Universal Robots PolyScope program: mansion.urp

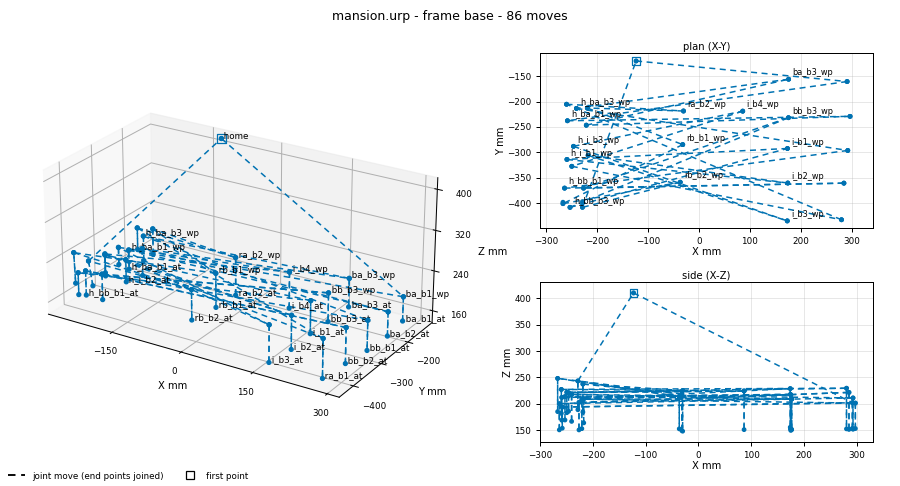
[picture p0: tool path of mansion.urp in frame base, 86 of 86 moves have a stored position in this frame; points joined in program order, loops and branches not executed]
Program mansion (installation=default directory=/programs/ITER createdIn=5.3.1.64192 lastSavedIn=5.3.1.64192 robotSerialNumber=20195300365)
Calibrated DH parameters: a=[-0.000093, -0.190649, -0.212673, 0.000091, -0.000205, 0]; d=[0.151591, 44.061648, -42.488068, -1.442789, 0.085322, 0.091911]; alpha=[1.570082, -0.003447, 0.007513, 1.572293, -1.571904, 0]; deltaTheta=[0, -0.672656, 0.728185, -0.055522, 0.000005, 0]
Robot Program (runOnlyOnce=true)
  URCap Gripper Activate (Robotiq_Grippers, Robotiq Inc.) dataModel(ResetAndActivateKey=false)
  URCap Gripper (Robotiq_Grippers, Robotiq Inc.) dataModel(position=50.0, force=100.0, speed=100.0, positionInDouble=50.0, forceInDouble=100.0, speedInDouble=100.0, slaveIds=[9], blocking=true)
  MoveJ speed 60 deg/s, acceleration 80 deg/s^2 (useActiveTCP=true) feature=Base
    Waypoint home: TCP in base x=-122.926 y=-120.377 z=410.038 mm, rx=2.273 ry=2.1657 rz=-0.0264 rad; joints [-85.876, -57.16, -80.452, -131.626, 89.649, -263.131] deg
  Folder Base_A
    MoveJ speed 60 deg/s, acceleration 80 deg/s^2 (useActiveTCP=true) feature=Base
      Waypoint ba_b1_wp: TCP in base x=291.339 y=-160.763 z=202.267 mm, rx=2.2196 ry=2.1634 rz=-0.046 rad; joints [-5.134, -97.09, -111.302, -60.85, 87.435, -183.275] deg
      Waypoint ba_b1_at: TCP in base x=291.327 y=-160.782 z=153.554 mm, rx=2.2196 ry=2.1633 rz=-0.046 rad; joints [-5.155, -104.362, -118.201, -46.683, 87.36, -183.222] deg
      URCap Gripper (Robotiq_Grippers, Robotiq Inc.) dataModel(position=100.0, force=100.0, speed=100.0, positionInDouble=100.0, forceInDouble=100.0, speedInDouble=100.0, slaveIds=[9], blocking=true)
      Waypoint ba_b1_wp: TCP in base x=291.339 y=-160.763 z=202.267 mm, rx=2.2196 ry=2.1634 rz=-0.046 rad; joints [-5.134, -97.09, -111.302, -60.85, 87.435, -183.275] deg
      Waypoint h_ba_b1_wp: TCP in base x=-257.858 y=-237.79 z=193.998 mm, rx=-3.1287 ry=0.0473 rz=-0.0059 rad; joints [-115.618, -102.966, -105.931, -61.783, 90.175, -203.494] deg
      Waypoint h_ba_b1_at: TCP in base x=-257.856 y=-237.787 z=153.878 mm, rx=-3.1287 ry=0.0473 rz=-0.006 rad; joints [-115.632, -108.549, -111.296, -50.837, 90.123, -203.451] deg
      URCap Gripper (Robotiq_Grippers, Robotiq Inc.) dataModel(position=50.0, force=100.0, speed=100.0, positionInDouble=50.0, forceInDouble=100.0, speedInDouble=100.0, slaveIds=[9], blocking=true)
      Waypoint h_ba_b1_wp: TCP in base x=-257.858 y=-237.79 z=193.998 mm, rx=-3.1287 ry=0.0473 rz=-0.0059 rad; joints [-115.618, -102.966, -105.931, -61.783, 90.175, -203.494] deg
    MoveJ speed 60 deg/s, acceleration 80 deg/s^2 (useActiveTCP=true) feature=Base
      Waypoint ba_b2_wp: TCP in base x=297.099 y=-229.137 z=201.509 mm, rx=2.2534 ry=2.1854 rz=-0.0426 rad; joints [-17.056, -107.569, -97.554, -65.462, 88.854, -194.942] deg
      Waypoint ba_b2_at: TCP in base x=297.093 y=-229.143 z=153.246 mm, rx=2.2534 ry=2.1854 rz=-0.0427 rad; joints [-17.073, -113.534, -103.963, -53.09, 88.799, -194.893] deg
      URCap Gripper (Robotiq_Grippers, Robotiq Inc.) dataModel(position=100.0, force=100.0, speed=100.0, positionInDouble=100.0, forceInDouble=100.0, speedInDouble=100.0, slaveIds=[9], blocking=true)
      Waypoint ba_b2_wp: TCP in base x=297.099 y=-229.137 z=201.509 mm, rx=2.2534 ry=2.1854 rz=-0.0426 rad; joints [-17.056, -107.569, -97.554, -65.462, 88.854, -194.942] deg
      Waypoint h_ba_b2_wp: TCP in base x=-220.82 y=-246.483 z=208.907 mm, rx=-3.1272 ry=0.0669 rz=0.002 rad; joints [-108.726, -96.552, -109.252, -64.858, 89.998, -195.885] deg
      Waypoint h_ba_b2_at: TCP in base x=-220.812 y=-246.497 z=153.058 mm, rx=-3.1273 ry=0.0669 rz=0.002 rad; joints [-108.744, -104.469, -117.433, -48.758, 89.918, -195.821] deg
      URCap Gripper (Robotiq_Grippers, Robotiq Inc.) dataModel(position=50.0, force=100.0, speed=100.0, positionInDouble=50.0, forceInDouble=100.0, speedInDouble=100.0, slaveIds=[9], blocking=true)
      Waypoint h_ba_b2_wp: TCP in base x=-220.82 y=-246.483 z=208.907 mm, rx=-3.1272 ry=0.0669 rz=0.002 rad; joints [-108.726, -96.552, -109.252, -64.858, 89.998, -195.885] deg
    MoveJ speed 60 deg/s, acceleration 80 deg/s^2 (useActiveTCP=true) feature=Base
      Waypoint ba_b3_wp: TCP in base x=176.479 y=-156.192 z=208.942 mm, rx=2.1987 ry=2.1726 rz=-0.0159 rad; joints [-7.147, -67.928, -134.317, -65.798, 88.131, -186.073] deg
      Waypoint ba_b3_at: TCP in base x=176.475 y=-156.198 z=150.955 mm, rx=2.1987 ry=2.1726 rz=-0.0159 rad; joints [-7.184, -79.69, -145.938, -42.419, 87.997, -185.98] deg
      URCap Gripper (Robotiq_Grippers, Robotiq Inc.) dataModel(position=100.0, force=100.0, speed=100.0, positionInDouble=100.0, forceInDouble=100.0, speedInDouble=100.0, slaveIds=[9], blocking=true)
      Waypoint ba_b3_wp: TCP in base x=176.479 y=-156.192 z=208.942 mm, rx=2.1987 ry=2.1726 rz=-0.0159 rad; joints [-7.147, -67.928, -134.317, -65.798, 88.131, -186.073] deg
      Waypoint h_ba_b3_wp: TCP in base x=-240.197 y=-213.51 z=217.855 mm, rx=2.242 ry=2.1952 rz=0.0362 rad; joints [-114.806, -93.519, -109.8, -67.774, 90.981, -293.227] deg
      Waypoint h_ba_b3_at: TCP in base x=-240.199 y=-213.502 z=166.817 mm, rx=2.242 ry=2.1953 rz=0.0361 rad; joints [-114.828, -100.186, -118.047, -52.858, 90.91, -293.168] deg
      URCap Gripper (Robotiq_Grippers, Robotiq Inc.) dataModel(position=50.0, force=100.0, speed=100.0, positionInDouble=50.0, forceInDouble=100.0, speedInDouble=100.0, slaveIds=[9], blocking=true)
      Waypoint h_ba_b3_wp: TCP in base x=-240.197 y=-213.51 z=217.855 mm, rx=2.242 ry=2.1952 rz=0.0362 rad; joints [-114.806, -93.519, -109.8, -67.774, 90.981, -293.227] deg
  Folder Base_B
    MoveJ speed 60 deg/s, acceleration 80 deg/s^2 (useActiveTCP=true) feature=Base
      Waypoint bb_b1_wp: TCP in base x=292.658 y=-296.109 z=211.213 mm, rx=2.2199 ry=2.2113 rz=-0.0547 rad; joints [-26.688, -116.102, -82.488, -71.567, 88.238, -206.181] deg
      Waypoint bb_b1_at: TCP in base x=292.645 y=-296.127 z=151.887 mm, rx=2.2199 ry=2.2112 rz=-0.0548 rad; joints [-26.711, -122.1, -90.484, -57.573, 88.188, -206.122] deg
      URCap Gripper (Robotiq_Grippers, Robotiq Inc.) dataModel(position=100.0, force=100.0, speed=100.0, positionInDouble=100.0, forceInDouble=100.0, speedInDouble=100.0, slaveIds=[9], blocking=true)
      Waypoint bb_b1_wp: TCP in base x=292.658 y=-296.109 z=211.213 mm, rx=2.2199 ry=2.2113 rz=-0.0547 rad; joints [-26.688, -116.102, -82.488, -71.567, 88.238, -206.181] deg
      Waypoint h_bb_b1_wp: TCP in base x=-263.499 y=-370.068 z=200.329 mm, rx=-3.0828 ry=0.0524 rz=-0.0261 rad; joints [-108.781, -127.406, -65.833, -80.171, 90.182, -196.637] deg
      Waypoint h_bb_b1_at: TCP in base x=-263.484 y=-370.083 z=150.732 mm, rx=-3.0828 ry=0.0523 rz=-0.026 rad; joints [-108.797, -131.383, -72.897, -69.13, 90.158, -196.59] deg
      URCap Gripper (Robotiq_Grippers, Robotiq Inc.) dataModel(position=50.0, force=100.0, speed=100.0, positionInDouble=50.0, forceInDouble=100.0, speedInDouble=100.0, slaveIds=[9], blocking=true)
      Waypoint h_bb_b1_wp: TCP in base x=-263.499 y=-370.068 z=200.329 mm, rx=-3.0828 ry=0.0524 rz=-0.0261 rad; joints [-108.781, -127.406, -65.833, -80.171, 90.182, -196.637] deg
    MoveJ speed 60 deg/s, acceleration 80 deg/s^2 (useActiveTCP=true) feature=Base
      Waypoint bb_b2_wp: TCP in base x=285.029 y=-360.313 z=221.676 mm, rx=2.2402 ry=2.1488 rz=-0.0282 rad; joints [-34.898, -125.685, -65.053, -77.312, 88.836, -212.332] deg
      Waypoint bb_b2_at: TCP in base x=285.033 y=-360.322 z=151.608 mm, rx=2.2401 ry=2.1488 rz=-0.028 rad; joints [-34.925, -131.234, -75.256, -61.556, 88.801, -212.266] deg
      URCap Gripper (Robotiq_Grippers, Robotiq Inc.) dataModel(position=100.0, force=100.0, speed=100.0, positionInDouble=100.0, forceInDouble=100.0, speedInDouble=100.0, slaveIds=[9], blocking=true)
      Waypoint bb_b2_wp: TCP in base x=285.029 y=-360.313 z=221.676 mm, rx=2.2402 ry=2.1488 rz=-0.0282 rad; joints [-34.898, -125.685, -65.053, -77.312, 88.836, -212.332] deg
      Waypoint h_bb_b2_wp: TCP in base x=-226.231 y=-370.058 z=202.804 mm, rx=-3.101 ry=0.0514 rz=-0.0119 rad; joints [-103.98, -121.699, -75.13, -75.447, 90.191, -191.835] deg
      Waypoint h_bb_b2_at: TCP in base x=-226.246 y=-370.053 z=150.663 mm, rx=-3.101 ry=0.0514 rz=-0.0119 rad; joints [-104.001, -126.505, -82.189, -63.582, 90.158, -191.786] deg
      URCap Gripper (Robotiq_Grippers, Robotiq Inc.) dataModel(position=50.0, force=100.0, speed=100.0, positionInDouble=50.0, forceInDouble=100.0, speedInDouble=100.0, slaveIds=[9], blocking=true)
      Waypoint h_bb_b2_wp: TCP in base x=-226.231 y=-370.058 z=202.804 mm, rx=-3.101 ry=0.0514 rz=-0.0119 rad; joints [-103.98, -121.699, -75.13, -75.447, 90.191, -191.835] deg
    MoveJ speed 60 deg/s, acceleration 80 deg/s^2 (useActiveTCP=true) feature=Base
      Waypoint bb_b3_wp: TCP in base x=176.16 y=-231.769 z=209.637 mm, rx=-2.2431 ry=-2.1874 rz=-0.0349 rad; joints [-26.842, -86.447, -119.81, -63.708, 91.685, -204.985] deg
      Waypoint bb_b3_at: TCP in base x=176.163 y=-231.779 z=151.997 mm, rx=-2.2432 ry=-2.1874 rz=-0.0349 rad; joints [-26.868, -95.964, -129.106, -44.891, 91.583, -204.91] deg
      URCap Gripper (Robotiq_Grippers, Robotiq Inc.) dataModel(position=100.0, force=100.0, speed=100.0, positionInDouble=100.0, forceInDouble=100.0, speedInDouble=100.0, slaveIds=[9], blocking=true)
      Waypoint bb_b3_wp: TCP in base x=176.16 y=-231.769 z=209.637 mm, rx=-2.2431 ry=-2.1874 rz=-0.0349 rad; joints [-26.842, -86.447, -119.81, -63.708, 91.685, -204.985] deg
      Waypoint h_bb_b3_wp: TCP in base x=-252.791 y=-407.786 z=213.756 mm, rx=2.2404 ry=2.1812 rz=0.0538 rad; joints [-106.357, -133.377, -52.558, -85.313, 91.957, -284.711] deg
      Waypoint h_bb_b3_at: TCP in base x=-252.772 y=-407.793 z=169.415 mm, rx=2.2404 ry=2.1812 rz=0.0537 rad; joints [-106.375, -135.74, -60.423, -75.082, 91.946, -284.663] deg
      URCap Gripper (Robotiq_Grippers, Robotiq Inc.) dataModel(position=50.0, force=100.0, speed=100.0, positionInDouble=50.0, forceInDouble=100.0, speedInDouble=100.0, slaveIds=[9], blocking=true)
      Waypoint h_bb_b3_wp: TCP in base x=-252.791 y=-407.786 z=213.756 mm, rx=2.2404 ry=2.1812 rz=0.0538 rad; joints [-106.357, -133.377, -52.558, -85.313, 91.957, -284.711] deg
  Folder Interconnect
    MoveJ speed 60 deg/s, acceleration 80 deg/s^2 (useActiveTCP=true) feature=Base
      Waypoint i_b1_wp: TCP in base x=174.192 y=-292.235 z=217.966 mm, rx=2.2497 ry=2.1639 rz=-0.0066 rad; joints [-36.697, -97.49, -106.294, -65.059, 89.868, -214.094] deg
      Waypoint i_b1_at: TCP in base x=174.179 y=-292.238 z=152.33 mm, rx=2.2498 ry=2.1638 rz=-0.0066 rad; joints [-36.724, -106.455, -115.875, -46.513, 89.778, -214.022] deg
      URCap Gripper (Robotiq_Grippers, Robotiq Inc.) dataModel(position=100.0, force=100.0, speed=100.0, positionInDouble=100.0, forceInDouble=100.0, speedInDouble=100.0, slaveIds=[9], blocking=true)
      Waypoint i_b1_wp: TCP in base x=174.192 y=-292.235 z=217.966 mm, rx=2.2497 ry=2.1639 rz=-0.0066 rad; joints [-36.697, -97.49, -106.294, -65.059, 89.868, -214.094] deg
      Waypoint h_i_b1_wp: TCP in base x=-258.783 y=-313.738 z=212.193 mm, rx=-3.0753 ry=0.0547 rz=-0.0056 rad; joints [-110.639, -114.762, -82.85, -75.951, 89.224, -198.304] deg
      Waypoint h_i_b1_at: TCP in base x=-258.784 y=-313.742 z=169.111 mm, rx=-3.0753 ry=0.0547 rz=-0.0057 rad; joints [-110.657, -118.67, -89.325, -65.57, 89.197, -198.259] deg
      URCap Gripper (Robotiq_Grippers, Robotiq Inc.) dataModel(position=50.0, force=100.0, speed=100.0, positionInDouble=50.0, forceInDouble=100.0, speedInDouble=100.0, slaveIds=[9], blocking=true)
      Waypoint h_i_b1_wp: TCP in base x=-258.783 y=-313.738 z=212.193 mm, rx=-3.0753 ry=0.0547 rz=-0.0056 rad; joints [-110.639, -114.762, -82.85, -75.951, 89.224, -198.304] deg
    MoveJ speed 60 deg/s, acceleration 80 deg/s^2 (useActiveTCP=true) feature=Base
      Waypoint i_b2_wp: TCP in base x=174.829 y=-360.086 z=217.004 mm, rx=2.2647 ry=2.1469 rz=-0.0178 rad; joints [-45.021, -111.703, -87.984, -69.069, 89.592, -221.659] deg
      Waypoint i_b2_at: TCP in base x=174.839 y=-360.085 z=149.76 mm, rx=2.2646 ry=2.147 rz=-0.0179 rad; joints [-45.043, -119.061, -97.021, -52.674, 89.527, -221.597] deg
      URCap Gripper (Robotiq_Grippers, Robotiq Inc.) dataModel(position=100.0, force=100.0, speed=100.0, positionInDouble=100.0, forceInDouble=100.0, speedInDouble=100.0, slaveIds=[9], blocking=true)
      Waypoint i_b2_wp: TCP in base x=174.829 y=-360.086 z=217.004 mm, rx=2.2647 ry=2.1469 rz=-0.0178 rad; joints [-45.021, -111.703, -87.984, -69.069, 89.592, -221.659] deg
      Waypoint h_i_b2_wp: TCP in base x=-217.209 y=-305.752 z=209.413 mm, rx=-3.1147 ry=0.0762 rz=0.0244 rad; joints [-104.846, -106.933, -95.847, -68.393, 89.071, -191.695] deg
      Waypoint h_i_b2_at: TCP in base x=-217.212 y=-305.747 z=163.983 mm, rx=-3.1147 ry=0.0762 rz=0.0244 rad; joints [-104.864, -112.08, -102.369, -56.726, 89.025, -191.646] deg
      URCap Gripper (Robotiq_Grippers, Robotiq Inc.) dataModel(position=50.0, force=100.0, speed=100.0, positionInDouble=50.0, forceInDouble=100.0, speedInDouble=100.0, slaveIds=[9], blocking=true)
      Waypoint h_i_b2_wp: TCP in base x=-217.209 y=-305.752 z=209.413 mm, rx=-3.1147 ry=0.0762 rz=0.0244 rad; joints [-104.846, -106.933, -95.847, -68.393, 89.071, -191.695] deg
    MoveJ speed 60 deg/s, acceleration 80 deg/s^2 (useActiveTCP=true) feature=Base
      Waypoint i_b3_wp: TCP in base x=173.862 y=-434.439 z=228.912 mm, rx=-2.2984 ry=-2.1342 rz=0.0077 rad; joints [-51.956, -128.706, -57.062, -84.438, 89.974, -227.564] deg
      Waypoint i_b3_at: TCP in base x=173.823 y=-434.448 z=155.772 mm, rx=-2.2985 ry=-2.1341 rz=0.0077 rad; joints [-51.993, -133.364, -69.125, -67.717, 89.949, -227.489] deg
      URCap Gripper (Robotiq_Grippers, Robotiq Inc.) dataModel(position=100.0, force=100.0, speed=100.0, positionInDouble=100.0, forceInDouble=100.0, speedInDouble=100.0, slaveIds=[9], blocking=true)
      Waypoint i_b3_wp: TCP in base x=173.862 y=-434.439 z=228.912 mm, rx=-2.2984 ry=-2.1342 rz=0.0077 rad; joints [-51.956, -128.706, -57.062, -84.438, 89.974, -227.564] deg
      Waypoint h_i_b3_wp: TCP in base x=-245.926 y=-287.976 z=221.138 mm, rx=2.2651 ry=2.1423 rz=0.0503 rad; joints [-110.984, -107.188, -92.208, -71.613, 92.308, -287.496] deg
      Waypoint b_i_b3_at: TCP in base x=-245.92 y=-287.99 z=185.909 mm, rx=2.265 ry=2.1423 rz=0.0502 rad; joints [-110.998, -110.532, -97.867, -62.605, 92.28, -287.458] deg
      URCap Gripper (Robotiq_Grippers, Robotiq Inc.) dataModel(position=50.0, force=100.0, speed=100.0, positionInDouble=50.0, forceInDouble=100.0, speedInDouble=100.0, slaveIds=[9], blocking=true)
      Waypoint h_i_b3_wp: TCP in base x=-245.926 y=-287.976 z=221.138 mm, rx=2.2651 ry=2.1423 rz=0.0503 rad; joints [-110.984, -107.188, -92.208, -71.613, 92.308, -287.496] deg
    MoveJ speed 60 deg/s, acceleration 80 deg/s^2 (useActiveTCP=true) feature=Base
      Waypoint i_b4_wp: TCP in base x=86.376 y=-218.928 z=224.266 mm, rx=2.2427 ry=2.1745 rz=0.0062 rad; joints [-35.112, -67.186, -129.953, -71.753, 90.433, -212.954] deg
      Waypoint i_b4_at: TCP in base x=86.374 y=-218.929 z=151.179 mm, rx=2.2427 ry=2.1745 rz=0.0061 rad; joints [-35.159, -80.22, -144.952, -43.721, 90.288, -212.837] deg
      URCap Gripper (Robotiq_Grippers, Robotiq Inc.) dataModel(position=100.0, force=100.0, speed=100.0, positionInDouble=100.0, forceInDouble=100.0, speedInDouble=100.0, slaveIds=[9], blocking=true)
      Waypoint i_b4_wp: TCP in base x=86.376 y=-218.928 z=224.266 mm, rx=2.2427 ry=2.1745 rz=0.0062 rad; joints [-35.112, -67.186, -129.953, -71.753, 90.433, -212.954] deg
      Waypoint h_i_b4_wp: TCP in base x=-249.299 y=-327.199 z=221.841 mm, rx=2.2374 ry=2.2006 rz=0.0433 rad; joints [-109.1, -114.821, -80.967, -75.483, 91.148, -287.896] deg
      Waypoint h_i_b4_at: TCP in base x=-249.283 y=-327.216 z=183.232 mm, rx=2.2374 ry=2.2006 rz=0.0433 rad; joints [-109.114, -117.988, -87.16, -66.124, 91.124, -287.854] deg
      URCap Gripper (Robotiq_Grippers, Robotiq Inc.) dataModel(position=50.0, force=100.0, speed=100.0, positionInDouble=50.0, forceInDouble=100.0, speedInDouble=100.0, slaveIds=[9], blocking=true)
      Waypoint h_i_b4_wp: TCP in base x=-249.299 y=-327.199 z=221.841 mm, rx=2.2374 ry=2.2006 rz=0.0433 rad; joints [-109.1, -114.821, -80.967, -75.483, 91.148, -287.896] deg
  Folder Roof_A
    MoveJ speed 60 deg/s, acceleration 80 deg/s^2 (useActiveTCP=true) feature=Base
      Waypoint ra_b1_wp: TCP in base x=280.355 y=-432.175 z=229.592 mm, rx=2.2498 ry=2.1383 rz=0.0086 rad; joints [-42.341, -144.4, -29.155, -94.202, 90.433, -219.411] deg
      Waypoint ra_b1_at: TCP in base x=280.345 y=-432.185 z=152.652 mm, rx=2.2498 ry=2.1383 rz=0.0087 rad; joints [-42.387, -145.97, -46.929, -74.856, 90.432, -219.319] deg
      URCap Gripper (Robotiq_Grippers, Robotiq Inc.) dataModel(position=100.0, force=100.0, speed=100.0, positionInDouble=100.0, forceInDouble=100.0, speedInDouble=100.0, slaveIds=[9], blocking=true)
      Waypoint ra_b1_wp: TCP in base x=280.355 y=-432.175 z=229.592 mm, rx=2.2498 ry=2.1383 rz=0.0086 rad; joints [-42.341, -144.4, -29.155, -94.202, 90.433, -219.411] deg
      Waypoint h_ra_b1_wp: TCP in base x=-259.638 y=-205.368 z=227.372 mm, rx=2.9429 ry=-0.031 rz=-0.0033 rad; joints [-120.289, -93.82, -112.087, -54.007, 95.739, -208.146] deg
      Waypoint h_ra_b1_at: TCP in base x=-259.633 y=-205.356 z=182.009 mm, rx=2.9429 ry=-0.031 rz=-0.0033 rad; joints [-120.304, -100.149, -119.184, -40.582, 95.664, -208.103] deg
      URCap Gripper (Robotiq_Grippers, Robotiq Inc.) dataModel(position=50.0, force=100.0, speed=100.0, positionInDouble=50.0, forceInDouble=100.0, speedInDouble=100.0, slaveIds=[9], blocking=true)
      Waypoint h_ra_b1_wp: TCP in base x=-259.638 y=-205.368 z=227.372 mm, rx=2.9429 ry=-0.031 rz=-0.0033 rad; joints [-120.289, -93.82, -112.087, -54.007, 95.739, -208.146] deg
    MoveJ speed 60 deg/s, acceleration 80 deg/s^2 (useActiveTCP=true) feature=Base
      Waypoint ra_b2_wp: TCP in base x=-29.938 y=-218.629 z=225.3 mm, rx=-2.2436 ry=-2.1936 rz=-0.0198 rad; joints [-62.186, -62.499, -131.394, -76.453, 91.059, -240.54] deg
      Waypoint ra_b2_at: TCP in base x=-29.954 y=-218.613 z=148.235 mm, rx=-2.2436 ry=-2.1934 rz=-0.0198 rad; joints [-62.247, -75.96, -148.106, -46.285, 90.919, -240.408] deg
      URCap Gripper (Robotiq_Grippers, Robotiq Inc.) dataModel(position=100.0, force=100.0, speed=100.0, positionInDouble=100.0, forceInDouble=100.0, speedInDouble=100.0, slaveIds=[9], blocking=true)
      Waypoint ra_b2_wp: TCP in base x=-29.938 y=-218.629 z=225.3 mm, rx=-2.2436 ry=-2.1936 rz=-0.0198 rad; joints [-62.186, -62.499, -131.394, -76.453, 91.059, -240.54] deg
      Waypoint h_ra_b2_wp: TCP in base x=-218.822 y=-212.79 z=237.473 mm, rx=0.0119 ry=3.1066 rz=-0.2822 rad; joints [-112.389, -86.229, -116.282, -58.23, 95.353, -381.095] deg
      Waypoint h_ra_b2_at: TCP in base x=-218.835 y=-212.79 z=184.432 mm, rx=0.012 ry=3.1067 rz=-0.2822 rad; joints [-112.412, -93.62, -125.525, -41.59, 95.263, -381.034] deg
      URCap Gripper (Robotiq_Grippers, Robotiq Inc.) dataModel(position=50.0, force=100.0, speed=100.0, positionInDouble=50.0, forceInDouble=100.0, speedInDouble=100.0, slaveIds=[9], blocking=true)
      Waypoint h_ra_b2_wp: TCP in base x=-218.822 y=-212.79 z=237.473 mm, rx=0.0119 ry=3.1066 rz=-0.2822 rad; joints [-112.389, -86.229, -116.282, -58.23, 95.353, -381.095] deg
  Folder Roof_B
    MoveJ speed 60 deg/s, acceleration 80 deg/s^2 (useActiveTCP=true) feature=Base
      Waypoint rb_b1_wp: TCP in base x=-31.427 y=-284.614 z=218.562 mm, rx=2.2451 ry=2.1882 rz=-0.0171 rad; joints [-69.272, -83.632, -119.946, -65.773, 89.911, -247.396] deg
      Waypoint rb_b1_at: TCP in base x=-31.436 y=-284.602 z=149.414 mm, rx=2.2452 ry=2.1882 rz=-0.017 rad; joints [-69.305, -95.054, -131.489, -42.815, 89.791, -247.308] deg
      URCap Gripper (Robotiq_Grippers, Robotiq Inc.) dataModel(position=100.0, force=100.0, speed=100.0, positionInDouble=100.0, forceInDouble=100.0, speedInDouble=100.0, slaveIds=[9], blocking=true)
      Waypoint rb_b1_wp: TCP in base x=-31.427 y=-284.614 z=218.562 mm, rx=2.2451 ry=2.1882 rz=-0.0171 rad; joints [-69.272, -83.632, -119.946, -65.773, 89.911, -247.396] deg
      Waypoint h_rb_b1_wp: TCP in base x=-266.628 y=-400.606 z=248.259 mm, rx=-2.9221 ry=0.0608 rz=-0.0496 rad; joints [-107.509, -142.729, -21.88, -117.881, 88.571, -195.052] deg
      Waypoint h_rb_b1_at: TCP in base x=-266.631 y=-397.735 z=185.295 mm, rx=-2.9221 ry=0.0608 rz=-0.0498 rad; joints [-107.672, -139.156, -45.769, -97.57, 88.599, -195.057] deg
      URCap Gripper (Robotiq_Grippers, Robotiq Inc.) dataModel(position=50.0, force=100.0, speed=100.0, positionInDouble=50.0, forceInDouble=100.0, speedInDouble=100.0, slaveIds=[9], blocking=true)
      Waypoint h_rb_b1_wp: TCP in base x=-266.628 y=-400.606 z=248.259 mm, rx=-2.9221 ry=0.0608 rz=-0.0496 rad; joints [-107.509, -142.729, -21.88, -117.881, 88.571, -195.052] deg
    MoveJ speed 60 deg/s, acceleration 80 deg/s^2 (useActiveTCP=true) feature=Base
      Waypoint rb_b2_wp: TCP in base x=-36.381 y=-358.469 z=213.765 mm, rx=-2.2634 ry=-2.1742 rz=-0.0315 rad; joints [-74.964, -103.256, -99.679, -67.697, 91.219, -252.317] deg
      Waypoint rb_b2_at: TCP in base x=-36.369 y=-358.47 z=152.678 mm, rx=-2.2633 ry=-2.1743 rz=-0.0315 rad; joints [-74.985, -110.842, -108.306, -51.483, 91.149, -252.255] deg
      URCap Gripper (Robotiq_Grippers, Robotiq Inc.) dataModel(position=100.0, force=100.0, speed=100.0, positionInDouble=100.0, forceInDouble=100.0, speedInDouble=100.0, slaveIds=[9], blocking=true)
      Waypoint rb_b2_wp: TCP in base x=-36.381 y=-358.469 z=213.765 mm, rx=-2.2634 ry=-2.1742 rz=-0.0315 rad; joints [-74.964, -103.256, -99.679, -67.697, 91.219, -252.317] deg
      Waypoint h_rb_b2_wp: TCP in base x=-228.341 y=-407.823 z=243.4 mm, rx=-2.9484 ry=0.091 rz=-0.0234 rad; joints [-102.754, -134.315, -39.474, -107.104, 89.06, -189.115] deg
      Waypoint h_rb_b2_at: TCP in base x=-228.326 y=-396.503 z=188.908 mm, rx=-2.9484 ry=0.091 rz=-0.0233 rad; joints [-103.117, -131.694, -58.874, -90.32, 89.017, -189.341] deg
      URCap Gripper (Robotiq_Grippers, Robotiq Inc.) dataModel(position=50.0, force=100.0, speed=100.0, positionInDouble=50.0, forceInDouble=100.0, speedInDouble=100.0, slaveIds=[9], blocking=true)
      Waypoint h_rb_b2_wp: TCP in base x=-228.341 y=-407.823 z=243.4 mm, rx=-2.9484 ry=0.091 rz=-0.0234 rad; joints [-102.754, -134.315, -39.474, -107.104, 89.06, -189.115] deg
  MoveJ speed 60 deg/s, acceleration 80 deg/s^2 (useActiveTCP=true) feature=Base
    Waypoint home: TCP in base x=-122.926 y=-120.377 z=410.038 mm, rx=2.273 ry=2.1657 rz=-0.0264 rad; joints [-85.876, -57.16, -80.452, -131.626, 89.649, -263.131] deg
